PROGRAM MAIN
VAR 
END_VAR

Accuracy_Measurement();

END_PROGRAM

(* stored: Version 1.1.0.1, ProductVersion 3.1.4024.12
   POU MAIN: Id {97acbdd3-2ab4-4801-ab26-b5f1255e7431}, SpecialFunc None *)
